TYPE "FeedMachine_Alr"
VERSION : 0.1
// Block: FeedMachine_Alr
   STRUCT
      BrakeTimeOut : Bool;
      Ax : TAx_Speed_Alarms;
      Fan_M : MotorAlr;
   END_STRUCT;

END_TYPE
